PROGRAM POU
VAR
//	FB_BurnerControlEcoFlam : FB_BurnerControlEcoFlam;
//	FB_BurnerControlEcoFlamV2 : FB_BurnerControlEcoFlamV2;
//	FB_BurnerControlEcoFlamV3 : FB_BurnerControlEcoFlamV3;
//	FB_ContactorFBNO : FB_ContactorFBNO;
//	fb_contactorNonFB : FB_ContactorNonFB;
//	FB_Contactor1FB_ThermalRelay : FB_Contactor1FB_ThermalRelay;
//	FB_ContactorNonFB_ThermalRelay : FB_ContactorNonFB_ThermalRelay;
//	FB_ContactorNonFB_Flex_ThermalRelay : FB_ContactorNonFB_Flex_ThermalRelay;
//	FB_SingleCoilCylinder : FB_SingleCoilCylinder;
//	FB_DoubleCoilCylinder : FB_DoubleCoilCylinder;
//	fbsingletank : FB_SingleTank;
//	fbsingletankV0 : FB_SingleTankV0;
//	fbsingletankV1 : FB_SingleTankV1;
//	fbTankFourCompartments : FB_TankFourCompartments;
//	fbSingleTankV1 : FB_SingleTanksV1;
//	fbFillTank : FB_TankFill_2Cylinder;
//	fbMixer0 : FB_Mixer0;
 	bIsClose : BOOL;
END_VAR

//fbSingleTankV1.AssignIfill(iFill := fbFillTank);
//bIsClose := fbsingletankV1.Ref_iFill.IsClose;

END_PROGRAM

(* stored: Version 1.1.0.1, ProductVersion 3.1.4024.12
   POU POU: Id {72876a34-3061-4895-8343-255626024a2e}, SpecialFunc None *)
